PROGRAM PRG_1_PlcTask
VAR
	
	
END_VAR

(*Ethercat Diagnostics*)
//DIAGNOSTICS();

PRG_Motors_Test();

// Functionblock for PTP motion between different appertures
//PRG_Motion();

// Vacuum and differential pumping
PRG_GATT();
// Injector
PRG_INJ();

//PRG_VGP();

END_PROGRAM

(* stored: Version 1.1.0.1, ProductVersion 3.1.4022.18
   POU PRG_1_PlcTask: Id {974f2793-1abb-41d3-ab47-a860d1c380f6}, SpecialFunc None *)
